KUKA KRL program: CeadHmi.src, CeadHmi.dat

--- CeadHmi.src ---
&ACCESS RVO
&REL 235
&COMMENT Ansteuerung Micromaster Frequenzumrichter
&PARAM EDITMASK = *
&PARAM TEMPLATE = C:\KRC\Roboter\Template\ExpertSubmit
&PARAM DISKPATH = KRC:\R1\TP\CNCRobotics\CEAD
DEF CeadHmi(   )
DECL INT i
;************************************************
;              CNC Robotics Ltd
;              www.cncrobotics.co.uk
;************************************************
;     Contact: helpdesk@cncrobotics.co.uk
;     Date: 26/09/23
;     Version: 0.5.51
;************************************************
; Description: sps control specific for the HMI
; related to the CEAD Extruder.
;************************************************

IF iRotationOn THEN
   rHmiPrintSpeed = $VEL_ACT * 1000
ELSE
   rHmiPrintSpeed = 0
ENDIF

MT.nNoOfTests = 0
MT.rSumOfValues = 0.0

FOR i = 1 TO 10
   IF (rMTRPM[i] > 0) AND (MT.rDensity <> 0) AND (MT.rTestTime <> 0) AND (rMTRPM[i] <> 0) THEN
      MT.nNoOfTests = MT.nNoOfTests + 1
      MT.rSumOfValues = MT.rSumOfValues + ((1000 * rMTWeight[i] / MT.rDensity) / MT.rTestTime) / rMTRPM[i]
   ENDIF
ENDFOR

IF (MT.nNoOfTests > 0) AND (MT.nNoOfTests <> 0) THEN
   MT.rMaterialConstant = MT.rSumOfValues / MT.nNoOfTests
ENDIF

IF (nMTTestNumber <> nMTPrevTestNumber) AND (MT.rDensity <> 0) AND (MT.rTestTime <> 0) AND (rMTRPM[nMTTestNumber] <> 0) THEN
   rMTVolume = (1000 * rMTWeight[nMTTestNumber] / MT.rDensity)
   rMTVolPerSec = rMTVolume / MT.rTestTime
   IF rMTRPM[nMTTestNumber] > 0 THEN
      rMTVolPerSecPerRPM = rMTVolPerSec / rMTRPM[nMTTestNumber]
   ENDIF
   nMTPrevTestNumber = nMTTestNumber
ENDIF

IF $PRO_STATE1 <> #P_FREE THEN
   bHmiHeaters=FALSE
   bHmiRotation=FALSE
   bHmiTransport=FALSE
ENDIF

IF $PRO_STATE1 == #P_FREE THEN

   IF bHmiSpeed0 THEN
      rScrewSet_rpm = 0
      bHmiSpeed0 = FALSE
   ENDIF

   IF bHmiSetSpeed THEN
      rScrewSet_rpm = rHmiExtruderSetSpeed
      bHmiSetSpeed = FALSE
   ENDIF

   IF (bHmiPurge) THEN
      MsgDialog(nHmiPurgeAns,"This program will move to purge position and purge the extruder.","CEAD",,,,,,,"Cancel","Continue", FALSE, nRobotMsg, E_spsMsgOpt)
      bHmiPurge = FALSE
   ENDIF

   IF (nHmiPurgeAns == 1) THEN
      CWRITE($CMD,E_stat,E_mode,"RUN/R1/Purge()")
       CWRITE($CMD,E_stat,E_mode,"STOP 1")
      nHmiPurgeAns = 0
   ENDIF

   IF (bHmiSystemPurge) THEN
      MsgDialog(nHmiSystemPurgeAns,"This program will fully purge the material from the extruder.","CEAD",,,,,,,"Cancel","Continue", FALSE, nRobotMsg, E_spsMsgOpt)
      bHmiSystemPurge = FALSE
   ENDIF

   IF (nHmiSystemPurgeAns == 1) THEN
      CWRITE($CMD,E_stat,E_mode,"RUN/R1/SystemPurge()")
       CWRITE($CMD,E_stat,E_mode,"STOP 1")
      nHmiSystemPurgeAns = 0
   ENDIF

ENDIF


END

--- CeadHmi.dat ---
&ACCESS  RV
&COMMENT Ansteuerung Micromaster Frequenzumrichter
&PARAM EDITMASK = *
&PARAM TEMPLATE = C:\KRC\Roboter\Template\ExpertSubmit
&PARAM DISKPATH = KRC:\R1\TP\CNCRobotics\CEAD
&REL 235
DEFDAT  CEADHMI PUBLIC

;************************************************
;              CNC Robotics Ltd
;              www.cncrobotics.co.uk
;************************************************
;     Contact: helpdesk@cncrobotics.co.uk
;     Date: 01/03/23
;     Version: 0.0.26
;************************************************
; Description: Dat file to store data for the
; printer.
;************************************************

;Extruder control from HMI flags
GLOBAL BOOL bHmiHeaters=FALSE
GLOBAL BOOL bHmiRotation=FALSE
GLOBAL BOOL bHmiTransport=FALSE

;Process control from HMI
GLOBAL BOOL bProportionalSpeed=FALSE
GLOBAL REAL rUserPercentage=100.000
GLOBAL REAL rHmiExtruderPercent=100.000
GLOBAL REAL rUserPercentageAtLock=100.000
GLOBAL REAL rOVatLock=100.000
GLOBAL REAL rHmiExtruderSetSpeed=50.0000
GLOBAL BOOL bHmiSetSpeed=FALSE
GLOBAL BOOL bHmiSpeed0=FALSE
GLOBAL BOOL bPrevProportionalSpeed=FALSE
GLOBAL BOOL bProportionalSpeedActive=TRUE
GLOBAL BOOL bPrevHmiRotation=FALSE
GLOBAL BOOL bStopAll=FALSE

;Purge button control
GLOBAL BOOL bHmiPurge=FALSE
GLOBAL INT nHmiPurgeAns=0
GLOBAL BOOL bHmiSystemPurge=FALSE
GLOBAL INT nHmiSystemPurgeAns=0

;HMI Display variables
GLOBAL REAL rCurrentLayer=100.000
GLOBAL REAL rTotalLayer=100.000
GLOBAL REAL rHmiPrintSpeed=0.0

ENDDAT
